INTERFACE itfCommand

METHOD Abort : MC_Error
VAR_INPUT
END_VAR
END_METHOD

PROPERTY Active : BOOL
GET
END_GET
SET
END_SET
END_PROPERTY

PROPERTY Busy : BOOL
GET
END_GET
SET
END_SET
END_PROPERTY

PROPERTY Command : MC_COMMAND_REF
GET
END_GET
SET
END_SET
END_PROPERTY

PROPERTY CommandAborted : BOOL
GET
END_GET
SET
END_SET
END_PROPERTY

PROPERTY Done : BOOL
GET
END_GET
SET
END_SET
END_PROPERTY

PROPERTY Error : BOOL
GET
END_GET
SET
END_SET
END_PROPERTY

PROPERTY ErrorId : MC_Error
GET
END_GET
SET
END_SET
END_PROPERTY

PROPERTY ErrorID_Udint : MC_ErrorID_Udint
GET
END_GET
SET
END_SET
END_PROPERTY

METHOD Wait 		: MC_Error // This method only makes sense in the IEC 61499 environment
VAR_INPUT
	Timeout		 	: TIME;
	AbortOnTimeout 	: BOOL; 
END_VAR
END_METHOD

END_INTERFACE

(* stored: Version 1.1.0.1, ProductVersion 3.1.4024.12
   Itf itfCommand: Id {5250b5ec-8adf-4a00-a8b0-e8cc89f6a9c6}
   Method Abort: Id {8879ef62-d1fc-4963-9a0b-5d65ca893dfc}
   Property Active: Id {28d3f1ac-2954-4588-88c8-61f6009efa8a}
   Get Get: Id {806e3e01-33a9-40fe-9670-357da9401fc9}
   Set Set: Id {46ee662c-65d1-446f-9d57-afbc25c43d46}
   Property Busy: Id {2d01e143-2399-43b7-863d-4b77823a55ba}
   Get Get: Id {d6976065-c885-4cbb-b8c9-c2875a8cba7b}
   Set Set: Id {eb38f715-f05d-440e-aa70-09f4173b521e}
   Property Command: Id {b2c9129f-feea-4473-85af-65f70883686d}
   Get Get: Id {d6ee44cb-7fe5-4561-a37e-94e880a17bd7}
   Set Set: Id {d6311410-f905-4229-b495-2ede7327b20b}
   Property CommandAborted: Id {91876b81-59bc-4e52-aebe-267a3038d803}
   Get Get: Id {75eb28ad-b2ef-4c04-8ca2-499550f652ca}
   Set Set: Id {0b6776f9-bc70-462c-9f3a-b91e57af12ef}
   Property Done: Id {ec239c16-214a-498b-be65-26f3b537b8ab}
   Get Get: Id {20fe5caa-4d4d-4baf-a9e9-35dcda8e4892}
   Set Set: Id {f8495318-8cf1-4974-a3d2-1a67d942a25d}
   Property Error: Id {37174fd7-cfb9-413b-8287-816c0a92597d}
   Get Get: Id {c9d4009b-62ee-42bf-856c-721709d018f2}
   Set Set: Id {2252b00b-101e-49a2-839e-b45750b7874e}
   Property ErrorId: Id {0d123eec-51a7-4234-bde4-c57b670a2bb8}
   Get Get: Id {675f6d49-1f8f-40e0-a984-498b0cc48137}
   Set Set: Id {400d7b0d-76a7-4efd-b755-df4b05d6a3d8}
   Property ErrorID_Udint: Id {aee349c9-8e08-42b4-a06e-76e3836bdd5a}
   Get Get: Id {c94dcbf0-2042-45a2-b517-6c19825cb383}
   Set Set: Id {619ef6d4-d46d-48e9-b1e6-47ee389854a8}
   Method Wait: Id {7b416bd3-0e82-47f6-ac03-447772e7f86d} *)
